Yaskawa INFORM job: JGFFG.JBI

/JOB
//NAME JGFFG
//POS
///NPOS 0,0,0,0,0,0
//INST
///DATE 2023/11/06 16:25
///ATTR SC,RW,RJ
////FRAME ROBOT
///GROUP1 RB1,BS1
NOP
END
